(* PLC project SansNom, Inconnu SansNom 1 *)
(* stored: creationDateTime 2024-10-07T10:59:27, modificationDateTime 2024-11-13T16:58:54 *)

TYPE AW9523B_1 : STRUCT
  Address : BYTE := 16#00;
  Init : BOOL := False;
  P0_0 : In_Out := Input;
  P0_1 : In_Out := Input;
  P0_2 : In_Out := Input;
  P0_3 : In_Out := Input;
  P0_4 : In_Out := Input;
  P0_5 : In_Out := Input;
  P0_6 : In_Out := Input;
  P0_7 : In_Out := Input;
  P1_0 : In_Out := Input;
  P1_1 : In_Out := Input;
  P1_2 : In_Out := Input;
  P1_3 : In_Out := Input;
  P1_4 : In_Out := Input;
  P1_5 : In_Out := Input;
  P1_6 : In_Out := Input;
  P1_7 : In_Out := Input;
END_STRUCT;
END_TYPE

TYPE In_Out : (Input, Output) := Input;
END_TYPE

TYPE AW9523B_2 : STRUCT
  Address : BYTE := 16#00;
  Init : BOOL := False;
  P1 : BYTE := 2#00000000;
  P2 : BYTE := 2#00000000;
END_STRUCT;
END_TYPE

TYPE datatype1 : BOOL;
END_TYPE

TYPE RLY08 : STRUCT
  CurrentAdress : BYTE := 16#00;
  WantAddress : BYTE := 16#00;
END_STRUCT;
END_TYPE

PROGRAM Plus10
  VAR RETAIN
    Count : INT := 0;
  END_VAR
  VAR RETAIN
    BP AT %IX0.1 : BOOL := 0;
  END_VAR
  VAR
    Test0 : Test;
  END_VAR
  VAR RETAIN
    Test1 : BYTE := 16#FF;
    BP1 : BOOL;
    LED1 : BOOL;
  END_VAR
  VAR
    KM1 : BOOL;
    KM2 : BOOL;
    KM3 : BOOL;
    M4 : BOOL;
    L1 : BOOL;
    L2 : BOOL;
    L3 : BOOL;
    Q1 : BOOL;
    Q2 : BOOL;
    Q3 : BOOL;
  END_VAR

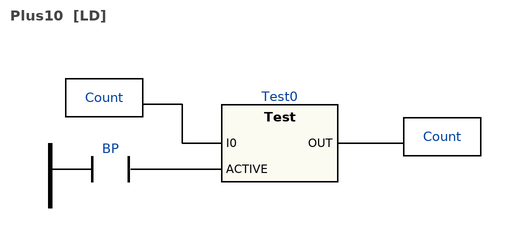
(* LD diagram, written out as Structured Text *)
Test0(I0 := Count, ACTIVE := BP);
Count := Test0.OUT;
END_PROGRAM

PROGRAM LED_BP
  VAR
    BP1 AT %IX0.0 : BOOL;
    LED AT %QX0.0 : BOOL;
  END_VAR

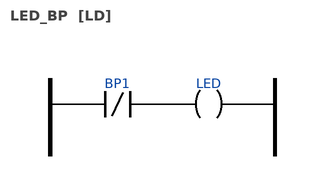
(* LD diagram, written out as Structured Text *)
LED := NOT BP1;
END_PROGRAM

FUNCTION function0 : BOOL
  VAR
    LocalVar0 : DINT;
  END_VAR

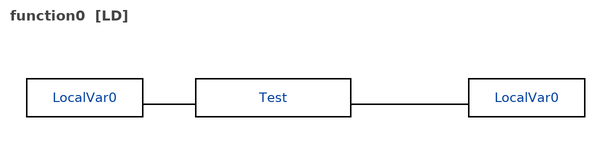
(* LD diagram, written out as Structured Text *)
Test := LocalVar0;
LocalVar0 := Test;
END_FUNCTION

PROGRAM NewBlock
  VAR
    DI_10 : DI_1;
    DI_11 : DINT;
    DQ_10 : DQ_1;
    DI_80 : DI_8;
    DQ_81 : DQ_8;
    RLY_10 : RLY_1;
    RLY_80 : RLY_8;
    Board1 : AW9523B_1;
    SET_ADDR0 : SET_ADDR;
  END_VAR
  VAR  (* added by the conversion: wires and edge detectors of the diagram *)
    _function054_OUT : BOOL;
  END_VAR

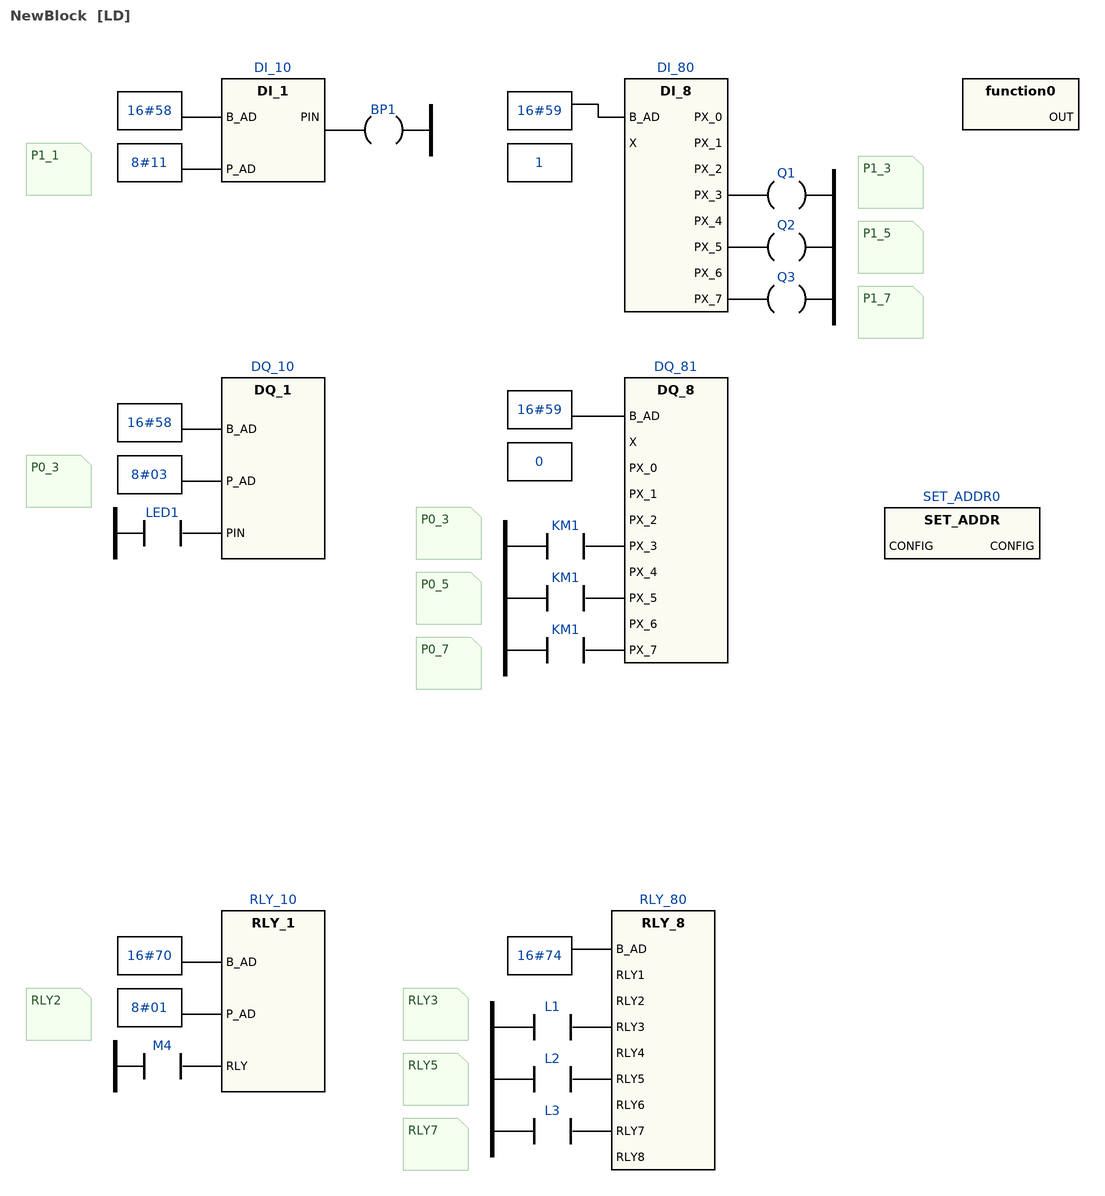
(* LD diagram, written out as Structured Text *)
DI_10(B_AD := 16#58, P_AD := 8#11);
BP1 := DI_10.PIN;
(* P1_1 *)
(* P1_3 *)
DI_80(B_AD := 16#59);
Q1 := DI_80.PX_3;
(* P1_5 *)
Q2 := DI_80.PX_5;
(* P1_7 *)
Q3 := DI_80.PX_7;
DQ_10(B_AD := 16#58, P_AD := 8#03, PIN := LED1);
DQ_81(B_AD := 16#59, PX_3 := KM1, PX_5 := KM1, PX_7 := KM1);
(* P0_3 *)
(* P0_3 *)
(* P0_5 *)
(* P0_7 *)
RLY_10(B_AD := 16#70, P_AD := 8#01, RLY := M4);
RLY_80(B_AD := 16#74, RLY3 := L1, RLY5 := L2, RLY7 := L3);
_function054_OUT := function0();
SET_ADDR0();
(* RLY2 *)
(* RLY3 *)
(* RLY3 *)
(* RLY5 *)
(* RLY7 *)
(* drawn but not wired to any output: 1, 0 *)
END_PROGRAM

FUNCTION_BLOCK functionBlock0
  VAR
    LocalVar0 : AW9523B_1;
  END_VAR

(* FBD diagram, written out as Structured Text *)
END_FUNCTION_BLOCK

PROGRAM program0
  VAR_EXTERNAL
    Board1 : AW9523B_1;
  END_VAR

            Board1
          
END_PROGRAM

CONFIGURATION Config0
  RESOURCE Res0 ON PLC
    VAR_GLOBAL
      Board1 : AW9523B_1;
    END_VAR
    TASK task0(INTERVAL := T#20ms, PRIORITY := 0);
    PROGRAM instance0 WITH task0 : Plus10;
  END_RESOURCE
END_CONFIGURATION
